(* CODESYS project Uebung4.library
   Company: ATS
   Title: Ueb4Lib
   Placeholder: Ueb4Lib
   Version: 1.0

Project tree, tasks and I/O mapping:
  libraries: Tc2_Standard, * (Beckhoff Automation GmbH); Tc2_System, * (Beckhoff Automation GmbH); Tc3_Module, * (Beckhoff Automation GmbH)
  DUTs/
  GVLs/
    global variables globe
  POUs/
    FiltAndInt/
      function block Integrator [ST]
      function block LowpassFilter [ST]
    Helper/
      function block EdgeDetectorWithDoubleTap [ST]
      function block GetTime [ST]
    Signals/
      function block PWMFunction [ST]
      function block SecondOrderLag [ST]
      function SinusFunction [ST]
      function SquareSignal [ST]
    program MAIN [ST]
  Version/
    global variables Global_Version
  VISUs/
  Uebung4.tmc
*)

// GVLs/globe

VAR_GLOBAL
	iglobCounter : INT;
	yellowButton AT %I* : BOOL;
	blueButton AT %I* : BOOL;
	greenLight AT %Q* : BOOL;
	redLight AT %Q* : BOOL;
	intUltrasonicSensor AT %I* : INT;
	iAnalogOutput AT %Q* : INT;
END_VAR

// Version/Global_Version
{attribute 'TcGenerated'}
// This function has been automatically generated from the project information.
VAR_GLOBAL CONSTANT
	{attribute 'const_non_replaced'}
	{attribute 'linkalways'}
	stLibVersion_Ueb4Lib : ST_LibVersion := (iMajor := 1, iMinor := 0, iBuild := 0, iRevision := 0, sVersion := '1.0');
END_VAR

// POUs/FiltAndInt/Integrator
FUNCTION_BLOCK Integrator

VAR_INPUT
	amplitude : REAL;
	cycleTicks : REAL; // Unter SYSTEM -> TASKS eingestellte ticks
END_VAR

VAR_OUTPUT
	area : REAL; // Fläche => Integral A(t)	
END_VAR

VAR
	tmpArea : REAL; // Die Fläche A(t-1)
	tmpAmplitude : REAL; // Die Amplitude P(t-1)
	T : REAL;// := ((10.0*1.0) / 1000.0);
END_VAR

	T  := ((cycleTicks*1.0) / 1000.0);
	area := tmpArea + ((tmpAmplitude + amplitude)/ 2.0) * T;
	tmpAmplitude := amplitude;
	tmpArea := area;

END_FUNCTION_BLOCK

// POUs/FiltAndInt/LowpassFilter
FUNCTION_BLOCK LowpassFilter

VAR_INPUT
	tau : REAL; // Ungefähr 0.1 testen
	input : REAL; // Signal
	cycleTicks : REAL; // Unter SYSTEM -> TASKS eingestellte ticks
END_VAR

VAR_OUTPUT
	output : REAL;
END_VAR

VAR
	T : REAL ;
	output_1 : REAL;
END_VAR

T :=  ((cycleTicks*1.0) / 1000.0);
output := (T/(T+tau)) * input + (tau/(T+tau)) * output_1;
output_1 := output;

END_FUNCTION_BLOCK

// POUs/Helper/EdgeDetectorWithDoubleTap
FUNCTION_BLOCK EdgeDetectorWithDoubleTap
VAR_INPUT
	inputValue : BOOL;
	timeBetweenTwoPresses : REAL; // in ms
END_VAR
VAR_OUTPUT
	risingEdge : BOOL;
	fallingEdge : BOOL;
	doubleTap : BOOL;
END_VAR
VAR
	oldSigVal : BOOL;
	timeCount : REAL;
	firstPress: BOOL := FALSE;
END_VAR

IF oldSigVal <> inputValue THEN
	IF inputValue = TRUE THEN
		IF firstPress = FALSE OR timeCount > timeBetweenTwoPresses THEN
		timeCount := 0.0;
		risingEdge := TRUE;
		firstPress := TRUE;
		ELSIF firstPress = TRUE AND timeCount < timeBetweenTwoPresses THEN
		doubleTap := TRUE;
		risingEdge := TRUE;
		timeCount := 0.0;
		END_IF
	ELSE
		risingEdge := FALSE;					
	END_IF
	fallingEdge := NOT risingEdge;
	oldSigVal := inputValue;
ELSE
	doubleTap := FALSE;
	risingEdge := FALSE;
	fallingEdge := FALSE;
END_IF
timeCount := timeCount + 1.0;

END_FUNCTION_BLOCK

// POUs/Helper/GetTime
FUNCTION_BLOCK GetTime
VAR_INPUT
	cycleTicks : REAL; // Unter SYSTEM -> TASKS eingestellte ticks
END_VAR
VAR_OUTPUT
	actTime : REAL;
END_VAR

VAR
	T : REAL;
	firstCall : BOOL := FALSE;
END_VAR

T  := ((cycleTicks*1.0) / 1000.0);
IF firstCall = FALSE THEN
	actTime := 0.0;
	firstCall := TRUE;
ELSE
	actTime := actTime + T;
END_IF

END_FUNCTION_BLOCK

// POUs/Signals/PWMFunction
FUNCTION_BLOCK PWMFunction
VAR_INPUT
	dutyCycle : REAL; // In % = t_ein / maxCount
	A : REAL; // Amplitude
	f : REAL; // Frequenz
	cycleTicks : REAL;
END_VAR

VAR_OUTPUT
	freqTooHigh : BOOL; //Verknüpfen mit roter LED
	pwm_Signal : REAL;
END_VAR

VAR
	T : REAL; // Zeit die das System braucht um den Funktionsblock einmal auzuführen
	fMax : REAL; // Maximale Frequnez die mit der TaskZeit erreicht werden kann
	counter : REAL;
	maxCount : REAL;
	t_ein : REAL;
END_VAR

// Taktzeit aus cycleTicks berechnen
T  := ((cycleTicks*1.0) / 1000.0);
IF T > 0.0 THEN
	fMax := 1.0 / T;
END_IF
IF f > fMax THEN
	freqTooHigh := TRUE;
	f := fMax;
END_IF
IF f > 0.0 THEN
	maxCount := (1.0 / f);
END_IF

t_ein := (dutyCycle / 100.0) * maxCount;

// Hauptzähler für Sägezahnrefernez
IF counter < maxCount THEN
	
	// PWM Generator
	IF t_ein >= counter THEN
		pwm_Signal := A;
	ELSE
		pwm_Signal := 0.0;
	END_IF
	counter := counter + T;
		
ELSIF counter >= maxCount THEN
	counter := 0.0;
END_IF

END_FUNCTION_BLOCK

// POUs/Signals/SecondOrderLag
FUNCTION_BLOCK SecondOrderLag

VAR_INPUT
	d : REAL; // Dämpfung
	w0 : REAL; // Eigenfrequnez
	input : REAL; // Eingangssignal
	cycleTicks : REAL; // Unter SYSTEM -> TASKS eingestellte ticks
END_VAR


VAR_OUTPUT
	output : REAL;
END_VAR


VAR
	T : REAL;
	a : REAL ;
	b : REAL ;
	c : REAL ;
	// Y(z) * a = U(z) * wo^2 + Y(z-1) * b - Y(z-2) * c
	output_1 : REAL;
	output_2 : REAL;
END_VAR

T := ((cycleTicks*1.0) / 1000.0);

//a  := (1.0/EXPT(T,2.0)) + (2.0/T)*d*w0  + EXPT(w0,2.0);
a := (1.0 / EXPT(T,2))+ 2.0 * d * w0 * (1.0/T)+EXPT(w0,2);
//b  := (2.0 / EXPT(T,2.0)) + (2.0/T) * d * w0;
b := (2.0/EXPT(T,2)) + (2.0 / T) * d * w0;
c  := (1.0/EXPT(T,2));

output := EXPT(w0,2) / a * input + b/a * output_1 - c/a * output_2;
output_2 := output_1;
output_1 := output;

END_FUNCTION_BLOCK

// POUs/Signals/SinusFunction
FUNCTION SinusFunction : REAL
VAR_INPUT
	A : REAL;
	yOffset : REAL;
	w : REAL;
	t : REAL;
END_VAR
VAR
END_VAR

SinusFunction := A * SIN(w*t) + yOffset;

END_FUNCTION

// POUs/Signals/SquareSignal
FUNCTION SquareSignal : REAL
VAR_INPUT
	yMin : REAL;
	yMAX : REAL;
	w : REAL;
	yOffset : REAL;
	t : REAL;
END_VAR
VAR
	reffSignal : REAL;
END_VAR

reffSignal := SIN(w*t) ;

IF(reffSignal > 0.0 ) THEN
	SquareSignal := yMAX + yOffset;
ELSIF reffSignal < 0.0 THEN
	SquareSignal := yMin + yOffset;
ELSE
	SquareSignal := 0.0;
END_IF

END_FUNCTION

// POUs/MAIN
PROGRAM MAIN
VAR
	blueButtonDetector : EdgeDetectorWithDoubleTap;
	yellowButtonDetector : EdgeDetectorWithDoubleTap;
	
	lowPass : LowpassFilter;
	lowPassSinus : LowpassFilter;
	secondOrder : SecondOrderLag;
	displayLowpass : REAL;
	btnToReal : REAL;
	displaySecondOrder : REAL;
	actTime : REAL := 0.0;
	sinus_Singal : REAL;
	square_Signal : REAL;
	pwm_Signal : REAL;
	sinus_SinlowPassSinusgal : REAL;
	integrate : Integrator;
	integrate2 : Integrator;
	risingEdgeLock : BOOL;
	rise : BOOL;
	displayIntegralOfSinus : REAL;
	displayIntegralOfSquare : REAL;
	displayLowpassSinus : REAL;
	currTime : GetTime;
END_VAR
VAR CONSTANT
	//T : REAL := 10.0 / 1000.0;
	omega : REAL := PI;
	ticks : REAL := 1.0;
END_VAR

blueButtonDetector(inputValue := blueButton, timeBetweenTwoPresses := 2000, risingEdge => rise);
IF rise THEN
	risingEdgeLock := TRUE;
END_IF


(*
Dürfen der Ausgang eines Funktionsblocks und die Variable auf die
dieser Ausgnag zugeweisen wird gleich heissen ???
*)
currTime(cycleTicks := ticks, actTime => actTime);
// Erzeugt einen Step beim Drücken eines Knopfes
IF blueButton OR yellowButton THEN
	btnToReal := 1.0;
ELSE
	btnToReal := 0.0;
END_IF
//displayLowpass auf Scope anzeigen
//lowPass(tau := 0.1,input := btnToReal,cycleTicks := ticks,output => displayLowpass);
//displaySecondOrder auf Scope anzeigen


//sinus_Singal := SinusFunction(A := 1.0, yOffset := 0.0, w := omega, t := actTime); 
square_Signal := SquareSignal(yMin := -1.0, yMax := 1.0, w := omega, yOffset := 0.0, t := actTime);
secondOrder(d := 0.001, w0 := 10, input := btnToReal,cycleTicks := ticks, output => displaySecondOrder);
//pwm_Signal := PWM_Function(cycleTicks := ticks, A := 1.0, t := actTime, f := 10.0,dutyCycle := 30.0);
//displayIntegralOfSinus auf Scope anzeigen
//integrate(amplitude := sinus_Singal,cycleTicks := ticks, area => displayIntegralOfSinus);
//displayIntegralOfSquare auf Scope anzeigen
// Müssen für diese zwei Zeilen wirklich 2 Instanzen von integrate erstellt werden?
//integrate2(amplitude := square_Signal,cycleTicks := ticks, area => displayIntegralOfSquare);
//sinus_SinlowPassSinusgal := SinusFunction(A := 1.0,yOffset := 0.0,w := 1.0 ,t := actTime);
//lowPassSinus(tau := 0.1,input := sinus_SinlowPassSinusgal,cycleTicks := ticks, output => displayLowpassSinus);

// Erstellen einer Bibliothek: https://infosys.beckhoff.com/index.php?content=../content/1031/tc3_plc_intro/9007203443996043.html&id=

END_PROGRAM
